Staubli VAL3: Page.pgx

program Page()
  local num l_nKey
begin
  //
  cls()
  nPage=1
  bExit=false
  do
    call RefreshPage()
    call RefreshBelt()
    l_nKey=getKey()
    call MainKey(l_nKey)
    delay(0)
  until bExit
  bExit=false
end
